PROGRAM Q6
VAR
	A : BOOL := TRUE;
	B : BOOL := FALSE;
	C : BOOL := FALSE;
END_VAR

// Result: C == TRUE

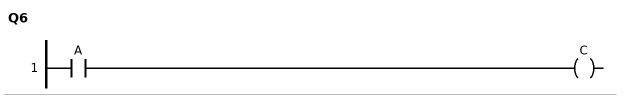
// NETWORK 1
C := A;

END_PROGRAM

(* stored: Version 1.1.0.1, ProductVersion 3.1.4024.12
   POU Q6: Id {8264a411-bdb2-415c-8c05-72587d002c47}, SpecialFunc None *)
